// TIA Portal V21 export
// export: Created 2026-09-06T18:39:46.4483401Z, ExportSetting WithDefaults, DisplayName Totally Integrated Automation Portal, DisplayVersion V21 Hotfix 1, DisplayName STEP 7 Professional, DisplayVersion V21, DisplayName STEP 7 CFC, DisplayVersion V21, DisplayName STEP 7 Safety, DisplayVersion V21, DisplayName Tech WebApplication, DisplayVersion V21, DisplayName WinCC Basic/Comfort/Advanced, DisplayVersion V21, DisplayName SIMATIC Visualization Architect, DisplayVersion V21, DisplayName WinCC Unified, DisplayVersion V21, DisplayName SIMATIC Visualization Architect, DisplayVersion V21
VAR_GLOBAL   // PLC tag table "Entradas_CPU_Local"
   STOP7 AT %I0.0 : Bool;   // Paragem Local / Botao Cogumelo de Paragem Geral (Contacto NF)
   START AT %I0.1 : Bool;   // Botao de Arranque do Sistema (Contacto NA)
   AVANCA AT %I0.2 : Bool;   // Botao Manual de Avanco do Cilindro Hidraulico (Contacto NA)
   RECUA AT %I0.3 : Bool;   // Botao Manual de Recuo do Cilindro Hidraulico (Contacto NA)
   FR1 AT %I0.4 : Bool;   // Disparo / Auxiliar do Rele Termico do Motor M1 (Contacto NF)
   FR2 AT %I0.5 : Bool;   // Disparo / Auxiliar do Rele Termico do Motor M2 (Contacto NF)
   FR3 AT %I0.6 : Bool;   // Disparo / Auxiliar do Rele Termico do Motor M3 (Contacto NF)
   FR4 AT %I0.7 : Bool;   // Disparo / Auxiliar do Rele Termico do Motor M4 (Contacto NF)
   FR5 AT %I1.0 : Bool;   // Disparo / Auxiliar do Rele Termico do Motor M5 (Contacto NF)
   FR6 AT %I1.1 : Bool;   // Disparo / Auxiliar do Rele Termico da Bomba M6 (Contacto NF)
   SEL_AUTO AT %I1.2 : Bool;   // Chave Seletora Auto/Manual - Posicao Automatico (Contacto NA)
   SEL_MANUAL AT %I1.3 : Bool;   // Chave Seletora Auto/Manual - Posicao Manual (Contacto NA)
   RESERVA_I1_4 AT %I1.4 : Bool;   // Reserva Tecnica Local CPU
   RESERVA_I1_5 AT %I1.5 : Bool;   // Reserva Tecnica Local CPU
END_VAR
